# EPICS substitutions: support/ebrick/2-2-3/iocBoot/iocebrick/ebrickDAC.substitutions
file ../../db/ebrDAC.db
{
pattern
{P         H       F       D       PREC    CH      PORT }

{ebrick:   ath01:  ana01:  ao01    3       0       ATHDAC }
{ebrick:   ath01:  ana01:  ao02    3       1       ATHDAC }
{ebrick:   ath01:  ana01:  ao03    3       2       ATHDAC }
{ebrick:   ath01:  ana01:  ao04    3       3       ATHDAC }

}
